PROGRAM PRG_IM6K2_PPM
VAR
    {attribute 'pytmc' := 'pv: IM6K2:PPM'}
    {attribute 'TcLinkTo' := '.fbGige.iIlluminatorINT := TIIB[IM6K2-EL4004-E7]^AO Outputs Channel 1^Analog output;
                              .fbGige.bGigePower := TIIB[IM6K2-EL2004-E3]^Channel 2^Output;
                              .fbPowerMeter.iVoltageINT := TIIB[IM6K2-EL3062-E6]^AI Standard Channel 1^Value;
                              .fbPowerMeter.fbThermoCouple.bError := TIIB[IM6K2-EL3314-E4]^TC Inputs Channel 1^Status^Error;
                              .fbPowerMeter.fbThermoCouple.bUnderrange := TIIB[IM6K2-EL3314-E4]^TC Inputs Channel 1^Status^Underrange;
                              .fbPowerMeter.fbThermoCouple.bOverrange := TIIB[IM6K2-EL3314-E4]^TC Inputs Channel 1^Status^Overrange;
                              .fbPowerMeter.fbThermoCouple.iRaw := TIIB[IM6K2-EL3314-E4]^TC Inputs Channel 1^Value;
                              .fbYagThermoCouple.bError := TIIB[IM6K2-EL3314-E4]^TC Inputs Channel 2^Status^Error;
                              .fbYagThermoCouple.bUnderrange := TIIB[IM6K2-EL3314-E4]^TC Inputs Channel 2^Status^Underrange;
                              .fbYagThermoCouple.bOverrange := TIIB[IM6K2-EL3314-E4]^TC Inputs Channel 2^Status^Overrange;
                              .fbYagThermoCouple.iRaw := TIIB[IM6K2-EL3314-E4]^TC Inputs Channel 2^Value'}
    fbIM6K2: FB_PPM;

    fbStateSetup: FB_StateSetupHelper;
    stDefault: ST_PositionState := (
        fVelocity := 12,
        bMoveOk := TRUE,
        bValid := TRUE
    );
END_VAR


fbStateSetup(stPositionState:=stDefault, bSetDefault:=TRUE);

fbStateSetup(stPositionState:=fbIM6K2.stOut, fPosition:=-8.61, sPmpsState:='IM6K2:PPM-OUT');
fbStateSetup(stPositionState:=fbIM6K2.stPower, fPosition:=-47.71, sPmpsState:='IM6K2:PPM-POWERMETER');
fbStateSetup(stPositionState:=fbIM6K2.stYag1, fPosition:=-71.71);
fbStateSetup(stPositionState:=fbIM6K2.stYag2, fPosition:=-97.72, sPmpsState:='IM6K2:PPM-YAG2');

CASE GVL.ePF2K2State OF
    E_WFS_STATES.TARGET1, E_WFS_STATES.TARGET2, E_WFS_STATES.TARGET3, E_WFS_STATES.TARGET4, E_WFS_STATES.TARGET5 :
        // Known state targets: allow less strict pmps
        fbIM6K2.stYag1.stPMPS.sPmpsState := 'IM6K2:PPM-YAG1_WFS_IN';
ELSE
    // Out, Unknown, or an unexpected state: full pmps
    fbIM6K2.stYag1.stPMPS.sPmpsState := 'IM6K2:PPM-YAG1';
END_CASE

fbIM6K2(
    fbFFHWO := GVL.fbFastFaultOutput2,
    fbArbiter := GVL.fbArbiter2,
    stYStage := Main.M24,
    sDeviceName := 'IM6K2:PPM',
    sTransitionKey := 'IM6K2:PPM-TRANSITION',
    bEnableMotion := TRUE,
    bEnableBeamParams := TRUE,
    bEnablePositionLimits := TRUE,
);

END_PROGRAM

(* stored: Version 1.1.0.1, ProductVersion 3.1.4022.18
   POU PRG_IM6K2_PPM: Id {b5662f22-bf30-4831-ae62-848249eb31cc}, SpecialFunc None *)
